(* CODESYS project BagFeedSequence.xml

Project tree, tasks and I/O mapping:
  function block BagFeedSequence [SFC]
*)

// BagFeedSequence
FUNCTION_BLOCK BagFeedSequence
VAR_INPUT
	Trigger: BOOL;
	FirstAdvanceComplete: BOOL;
	FirstRetractComplete: BOOL;
	RetryAdvanceComplete: BOOL;
	RetryRetractComplete: BOOL;
	BagOpen: BOOL;
	HeatSealClosed: BOOL;
	HeatSealOpened: BOOL;
END_VAR
VAR_OUTPUT
	BlowerOn: BOOL;
	FirstAdvance: BOOL;
	FirstRetract: BOOL;
	RetryAdvance: BOOL;
	RetryRetract: BOOL;
	FillIce: BOOL;
	CloseBag: BOOL;
	PresentBag: BOOL;	
	TearBag: BOOL;
	KickerRaised: BOOL;
END_VAR
VAR
	_attempts: UINT;
END_VAR

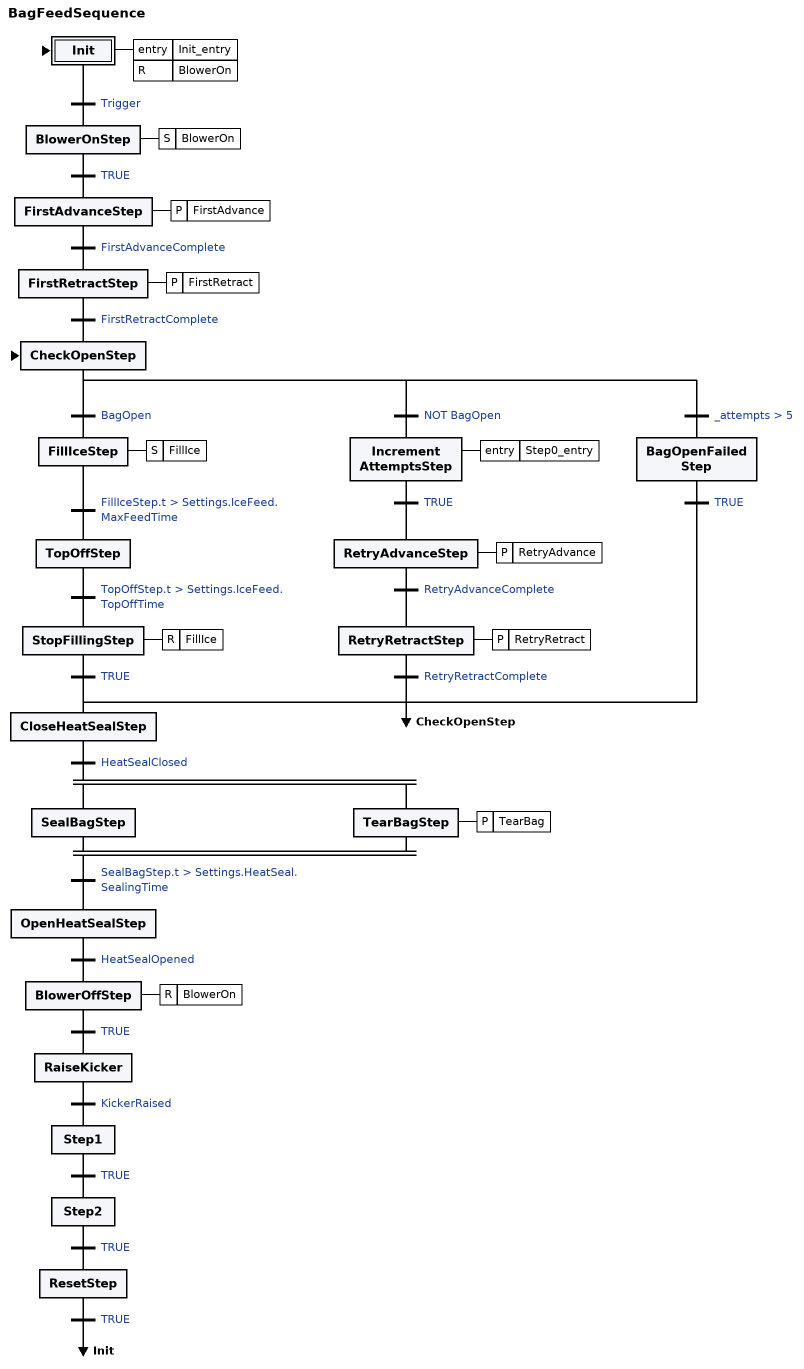
INITIAL_STEP Init:
    Init_entry(P1);  // entry action
    BlowerOn(R);
END_STEP
TRANSITION FROM Init TO BlowerOnStep
    := Trigger;
END_TRANSITION
STEP BlowerOnStep:
    BlowerOn(S);
END_STEP
TRANSITION FROM BlowerOnStep TO FirstAdvanceStep
    := TRUE;
END_TRANSITION
STEP FirstAdvanceStep:
    FirstAdvance(P);
END_STEP
TRANSITION FROM FirstAdvanceStep TO FirstRetractStep
    := FirstAdvanceComplete;
END_TRANSITION
STEP FirstRetractStep:
    FirstRetract(P);
END_STEP
TRANSITION FROM FirstRetractStep TO CheckOpenStep
    := FirstRetractComplete;
END_TRANSITION
STEP CheckOpenStep:
END_STEP
TRANSITION FROM CheckOpenStep TO FillIceStep
    := BagOpen;
END_TRANSITION
TRANSITION FROM CheckOpenStep TO IncrementAttemptsStep
    := NOT BagOpen;
END_TRANSITION
STEP IncrementAttemptsStep:
    Step0_entry(P1);  // entry action
END_STEP
TRANSITION FROM IncrementAttemptsStep TO RetryAdvanceStep
    := TRUE;
END_TRANSITION
STEP RetryAdvanceStep:
    RetryAdvance(P);
END_STEP
TRANSITION FROM RetryAdvanceStep TO RetryRetractStep
    := RetryAdvanceComplete;
END_TRANSITION
STEP RetryRetractStep:
    RetryRetract(P);
END_STEP
TRANSITION FROM RetryRetractStep TO CheckOpenStep
    := RetryRetractComplete;
END_TRANSITION
STEP FillIceStep:
    FillIce(S);
END_STEP
TRANSITION FROM FillIceStep TO TopOffStep
    := FillIceStep.t > Settings.IceFeed.MaxFeedTime;
END_TRANSITION
STEP TopOffStep:
END_STEP
TRANSITION FROM TopOffStep TO StopFillingStep
    := TopOffStep.t > Settings.IceFeed.TopOffTime;
END_TRANSITION
STEP StopFillingStep:
    FillIce(R);
END_STEP
TRANSITION FROM StopFillingStep TO CloseHeatSealStep
    := TRUE;
END_TRANSITION
TRANSITION FROM CheckOpenStep TO BagOpenFailedStep
    := _attempts > 5;
END_TRANSITION
STEP BagOpenFailedStep:
END_STEP
TRANSITION FROM BagOpenFailedStep TO CloseHeatSealStep
    := TRUE;
END_TRANSITION
STEP CloseHeatSealStep:
END_STEP
TRANSITION FROM CloseHeatSealStep TO (SealBagStep, TearBagStep)
    := HeatSealClosed;
END_TRANSITION
STEP SealBagStep:
END_STEP
STEP TearBagStep:
    TearBag(P);
END_STEP
TRANSITION FROM (SealBagStep, TearBagStep) TO OpenHeatSealStep
    := SealBagStep.t > Settings.HeatSeal.SealingTime;
END_TRANSITION
STEP OpenHeatSealStep:
END_STEP
TRANSITION FROM OpenHeatSealStep TO BlowerOffStep
    := HeatSealOpened;
END_TRANSITION
STEP BlowerOffStep:
    BlowerOn(R);
END_STEP
TRANSITION FROM BlowerOffStep TO RaiseKicker
    := TRUE;
END_TRANSITION
STEP RaiseKicker:
END_STEP
TRANSITION FROM RaiseKicker TO Step1
    := KickerRaised;
END_TRANSITION
STEP Step1:
END_STEP
TRANSITION FROM Step1 TO Step2
    := TRUE;
END_TRANSITION
STEP Step2:
END_STEP
TRANSITION FROM Step2 TO ResetStep
    := TRUE;
END_TRANSITION
STEP ResetStep:
END_STEP
TRANSITION FROM ResetStep TO Init
    := TRUE;
END_TRANSITION
// branch label SealBagBranch

END_FUNCTION_BLOCK
